TYPE ST_SafetyFeedback :
STRUCT
END_STRUCT
END_TYPE

(* stored: Version 1.1.0.1
   DUT ST_SafetyFeedback: Id {6e0330ba-8186-0b3e-1827-26396cd792da} *)
